Fanuc KAREL source: kt00254.KL

-- PROVISIONAL review KL for V1013-1; original PC SHA256 2026578bbaadf62336cbd8f818a4f6be8a600db8f77530bba069af31f2f33a77
-- Incomplete behavior may be omitted. Consult companion uncertainty JSON. Do not deploy.
PROGRAM KT00254
%NOLOCKGROUP
VAR
  OUT : INTEGER
-- UNRESOLVED_DECL H1 type=002017
-- UNRESOLVED_DECL Y2 type=002018
BEGIN
  -- UNRESOLVED_PC offsets 5-19; opcodes 2E,22,9D,33,B4
  -- UNRESOLVED_PC offsets 24-38; opcodes 2E,22,9D,33,B2
  -- UNRESOLVED_PC offsets 43-68; opcodes 22,9D,33,B3,22,9D,33,B1,47,23
  -- UNRESOLVED_PC offsets 73-77; opcodes 7F
END KT00254
